// TIA Portal project "Phase 1" (V15.1)

(* hardware
DEVICE "S71500/ET200MP-Station_1"  S7-1500 station
   slot 0: "Profilschiene_0"  6ES7 590-1***0-0AA0
   slot 1: "PLC_1"  CPU 1511-1 PN  6ES7 511-1AK00-0AB0  V1.8
   slot 2: "AI 8xU/I/RTD/TC ST_1"  AI 8xU/I/RTD/TC ST  6ES7 531-7KF00-0AB0  V2.0
   slot 3: "AI 8xU/I/RTD/TC ST_2"  AI 8xU/I/RTD/TC ST  6ES7 531-7KF00-0AB0  V2.0
   slot 4: "AI 8xU/I/RTD/TC ST_3"  AI 8xU/I/RTD/TC ST  6ES7 531-7KF00-0AB0  V2.0
   slot 5: "AI 8xU/I/RTD/TC ST_4"  AI 8xU/I/RTD/TC ST  6ES7 531-7KF00-0AB0  V2.0
   slot 6: "DI 16x24VDC BA_1"  DI 16x24VDC BA  6ES7 521-1BH10-0AA0  V1.0
DEVICE "HMI_1"  KTP700 Basic PN
   slot 0: "HMI_1"  KTP700 Basic PN  6AV2 123-2GB03-0AX0  15.1.0.0
   slot 1: "HMI_RT_1"  KTP700 Basic PN  6AV2 123-2GB03-0AX0  15.1.0.0
   slot 5: "HMI_1.IE_CP_1"  PROFINET Interface  15.0.1.0
      slot 1: "PROFINET Interface_1"  PROFINET Interface
         slot 1: "Port_1"  Port
*)

// ===== PLC "PLC_1"  CPU 1511-1 PN =====

VAR_GLOBAL   // PLC tag table "Standard-Variablentabelle"
   "LevelMeter" AT %IW30 : Word;
   "FlowMeter" AT %IW32 : Word;
   "Set_point" AT %IW34 : Word;
   "Norm_SP" AT %MD74 : Real;
   "PID_Output" AT %MD104 : Real;
   "Start" AT %I10.0 : Bool;
   "Fill_Valve" AT %QW30 : Word;
   "Start_Light" AT %Q10.0 : Bool;
   "Reset" AT %I10.1 : Bool;
   "Reset_Light" AT %Q10.1 : Bool;
   "On" AT %M2.1 : Bool;
   "Stop" AT %I10.2 : Bool;
   "Stop_Light" AT %Q10.2 : Bool;
   "PV_display" AT %QW36 : Word;
   "Setpoint_display" AT %QW34 : Word;
   "Setpoint_value" AT %MD200 : Real;
   "Process_value" AT %MD204 : Real;
   "Norm_PID_Output" AT %MD208 : Real;
   "Start_from_HMI" AT %M4.0 : Bool;
   "Stop_from_HMI" AT %M4.1 : Bool;
   "Reset_from_HMI" AT %M4.2 : Bool;
   "Start_flag" AT %M5.0 : Bool;
   "Reset_flag" AT %M5.1 : Bool;
   "Stop_flag" AT %M5.2 : Bool;
   "Switch" AT %M5.3 : Bool;
   "Set_form_HMI" AT %MW216 : Word;
   "Norm_level" AT %MD212 : Real;
   "Level_error_margin" AT %MD218 : Real;
   "High_level_threshold" AT %MD220 : Real;
   "Low_level_threshold" AT %MD222 : Real;
   "Digital alarms" AT %MW6 : Word;
   "Discharge valve" AT %QW32 : Word;
END_VAR

// folder: System blocks/Program resources

DATA_BLOCK "IEC_Timer_0_DB"   // DB4
{ S7_Optimized_Access := 'TRUE' }
AUTHOR : Simatic
FAMILY : IEC
NAME : IEC_TMR
VERSION : 1.0
// stored: InstanceOfName IEC_TIMER
"IEC_TIMER"
BEGIN
END_DATA_BLOCK

// folder: (top level)

FUNCTION "MHJ-PLC-Lab-Function-S71500" : Void   // FC9000, SCL
{ S7_Optimized_Access := 'TRUE' }
VERSION : 0.1
   VAR_TEMP
      Value : Byte;
      ForCounter : Int;
   END_VAR
   VAR CONSTANT
      Value_01_DW : DWord := 16#1223_5486;
      Value_02_DW : DWord := 16#A6C9_D1F5;
   END_VAR
BEGIN

   #Value:=PEEK(area := 16#82,
        dbNumber := 0,
        byteOffset := 511);
   #Value := #Value + 1;

   POKE(area := 16#82,
        dbNumber := 0,
        byteOffset := 511,
        value := #Value);

   POKE(area := 16#82,
        dbNumber := 0,
        byteOffset := 1016,
        value := #Value_01_DW);
   POKE(area := 16#82,
        dbNumber := 0,
        byteOffset := 1020,
        value := #Value_02_DW);

   FOR #ForCounter := 0 TO 63 DO
       #Value:=PEEK(area := 16#1,
            dbNumber := 0,
            byteOffset := #ForCounter);
       POKE(area := 16#81,
            dbNumber := 0,
            byteOffset := #ForCounter,
            value := #Value);
   END_FOR;
   #Value := PEEK(area := 16#1,
                  dbNumber := 0,
                  byteOffset := 512);
   POKE(area := 16#82,
        dbNumber := 0,
        byteOffset := 512,
        value := #Value);
END_FUNCTION

ORGANIZATION_BLOCK "Main"   // OB1, FBD, ProgramCycle
TITLE = "Main Program Sweep (Cycle)"
{ S7_Optimized_Access := 'TRUE' }
VERSION : 0.1
   VAR_INPUT
      Initial_Call : Bool;   // Initial call of this OB
      Remanence : Bool;   // =True, if remanent data are available
   END_VAR
BEGIN

REGION Network 1
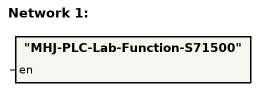
   "MHJ-PLC-Lab-Function-S71500"();
END_REGION
END_ORGANIZATION_BLOCK

ORGANIZATION_BLOCK "Cyclic interrupt"   // OB30, LAD, CyclicInterrupt
{ S7_Optimized_Access := 'TRUE' }
VERSION : 0.1
   VAR_INPUT
      Initial_Call : Bool;   // Initial call of this OB
      Event_Count : Int;   // Events discarded
   END_VAR
BEGIN

REGION Network 1
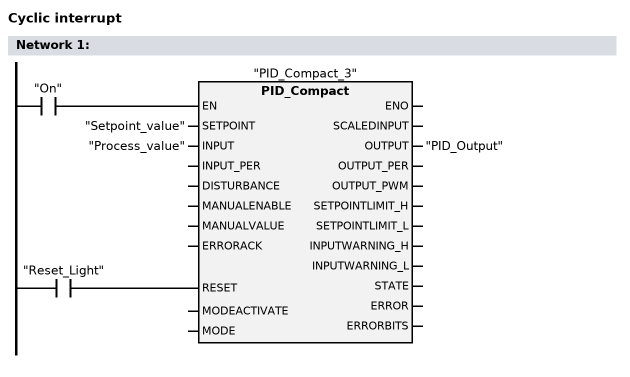
   IF "On" THEN
       "PID_Compact_3"(Setpoint := "Setpoint_value",   // PID_Compact
                       Input := "Process_value",
                       Reset := "Reset_Light",
                       Output => "PID_Output");
   END_IF;
END_REGION
END_ORGANIZATION_BLOCK

ORGANIZATION_BLOCK "Main_1"   // OB123, LAD, ProgramCycle
TITLE = "Main Program Sweep (Cycle)"
{ S7_Optimized_Access := 'TRUE' }
VERSION : 0.1
   VAR_INPUT
      Initial_Call : Bool;   // Initial call of this OB
      Remanence : Bool;   // =True, if remanent data are available
   END_VAR
BEGIN

REGION Network 1: Set point scale & display
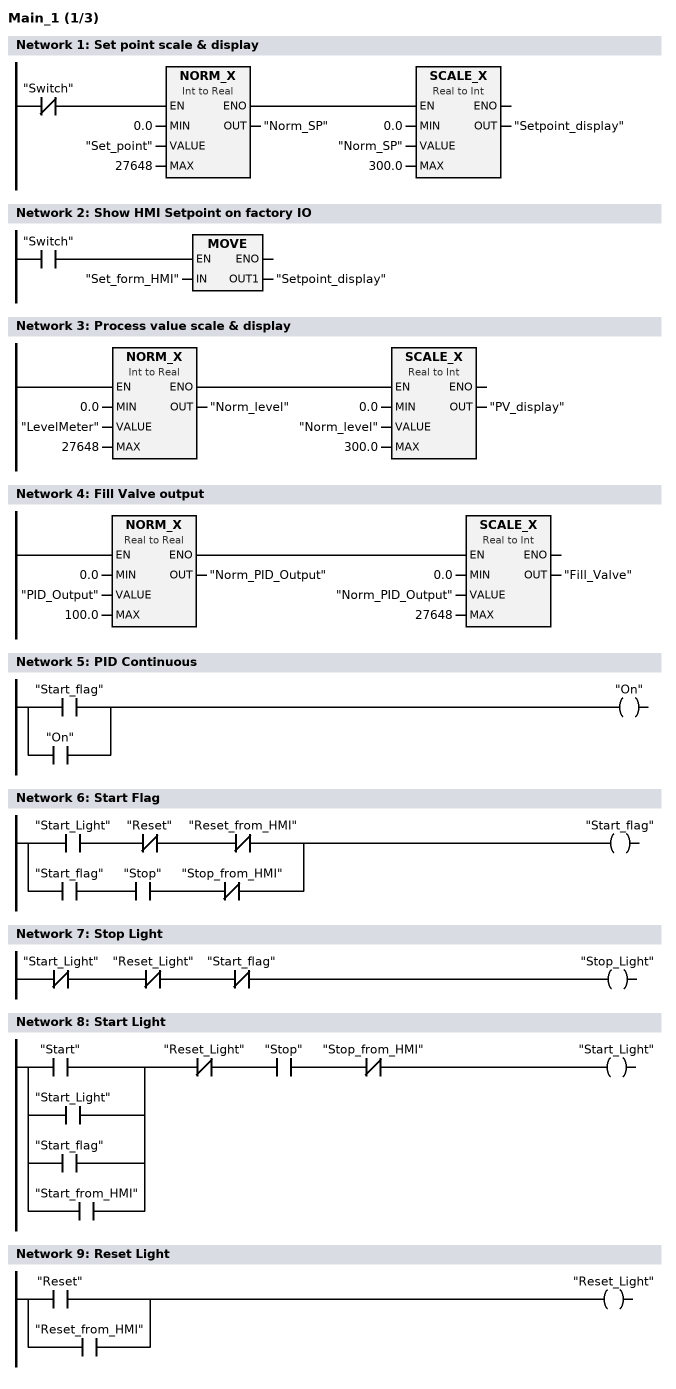
   RUNG wire#powerrail
      I_Contact( "Switch" )
      { S7_Templates := "[SrcType := Int, DestType := Real]" } Normalize(min := 0.0, value := "Set_point", max := 27648, out => "Norm_SP")
      { S7_Templates := "[SrcType := Real, DestType := Int]" } Scale(min := 0.0, value := "Norm_SP", max := 300.0, out => "Setpoint_display")
   END_RUNG
   // the same network as SCL:
   IF NOT "Switch" THEN
       "Norm_SP" := NORM_X(MIN := 0.0, VALUE := "Set_point", MAX := 27648);
       "Setpoint_display" := SCALE_X(MIN := 0.0, VALUE := "Norm_SP", MAX := 300.0);
   END_IF;
END_REGION

REGION Network 2: Show HMI Setpoint on factory IO
   RUNG wire#powerrail
      Contact( "Switch" )
      Move(in := "Set_form_HMI", out1 => "Setpoint_display")
   END_RUNG
   // the same network as SCL:
   IF "Switch" THEN "Setpoint_display" := "Set_form_HMI"; END_IF;
END_REGION

REGION Network 3: Process value scale & display
   RUNG wire#powerrail
      { S7_Templates := "[SrcType := Int, DestType := Real]" } Normalize(min := 0.0, value := "LevelMeter", max := 27648, out => "Norm_level")
      { S7_Templates := "[SrcType := Real, DestType := Int]" } Scale(min := 0.0, value := "Norm_level", max := 300.0, out => "PV_display")
   END_RUNG
   // the same network as SCL:
   "Norm_level" := NORM_X(MIN := 0.0, VALUE := "LevelMeter", MAX := 27648);
   "PV_display" := SCALE_X(MIN := 0.0, VALUE := "Norm_level", MAX := 300.0);
END_REGION

REGION Network 4: Fill Valve output
   RUNG wire#powerrail
      { S7_Templates := "[SrcType := Real, DestType := Real]" } Normalize(min := 0.0, value := "PID_Output", max := 100.0, out => "Norm_PID_Output")
      { S7_Templates := "[SrcType := Real, DestType := Int]" } Scale(min := 0.0, value := "Norm_PID_Output", max := 27648, out => "Fill_Valve")
   END_RUNG
   // the same network as SCL:
   "Norm_PID_Output" := NORM_X(MIN := 0.0, VALUE := "PID_Output", MAX := 100.0);
   "Fill_Valve" := SCALE_X(MIN := 0.0, VALUE := "Norm_PID_Output", MAX := 27648);
END_REGION

REGION Network 5: PID Continuous
   RUNG wire#powerrail
      Contact( "Start_flag" )
      wire#w1
      Coil( "On" )
   END_RUNG
   RUNG wire#powerrail
      Contact( "On" )
   END_RUNG wire#w1
   // the same network as SCL:
   "On" := "Start_flag" OR "On";
END_REGION

REGION Network 6: Start Flag
   RUNG wire#powerrail
      Contact( "Start_Light" )
      I_Contact( "Reset" )
      I_Contact( "Reset_from_HMI" )
      wire#w1
      Coil( "Start_flag" )
   END_RUNG
   RUNG wire#powerrail
      Contact( "Start_flag" )
      Contact( "Stop" )
      I_Contact( "Stop_from_HMI" )
   END_RUNG wire#w1
   // the same network as SCL:
   "Start_flag" := ("Start_Light" AND NOT "Reset" AND NOT "Reset_from_HMI") OR ("Start_flag" AND "Stop" AND NOT "Stop_from_HMI");
END_REGION

REGION Network 7: Stop Light
   RUNG wire#powerrail
      I_Contact( "Start_Light" )
      I_Contact( "Reset_Light" )
      I_Contact( "Start_flag" )
      Coil( "Stop_Light" )
   END_RUNG
   // the same network as SCL:
   "Stop_Light" := NOT "Start_Light" AND NOT "Reset_Light" AND NOT "Start_flag";
END_REGION

REGION Network 8: Start Light
   RUNG wire#powerrail
      Contact( "Start" )
      wire#w1
      I_Contact( "Reset_Light" )
      Contact( "Stop" )
      I_Contact( "Stop_from_HMI" )
      Coil( "Start_Light" )
   END_RUNG
   RUNG wire#powerrail
      Contact( "Start_Light" )
   END_RUNG wire#w1
   RUNG wire#powerrail
      Contact( "Start_flag" )
   END_RUNG wire#w1
   RUNG wire#powerrail
      Contact( "Start_from_HMI" )
   END_RUNG wire#w1
   // the same network as SCL:
   "Start_Light" := ("Start" OR "Start_Light" OR "Start_flag" OR "Start_from_HMI") AND NOT "Reset_Light" AND "Stop" AND NOT "Stop_from_HMI";
END_REGION

REGION Network 9: Reset Light
   RUNG wire#powerrail
      Contact( "Reset" )
      wire#w1
      Coil( "Reset_Light" )
   END_RUNG
   RUNG wire#powerrail
      Contact( "Reset_from_HMI" )
   END_RUNG wire#w1
   // the same network as SCL:
   "Reset_Light" := "Reset" OR "Reset_from_HMI";
END_REGION

REGION Network 10: Fill Valve Stop
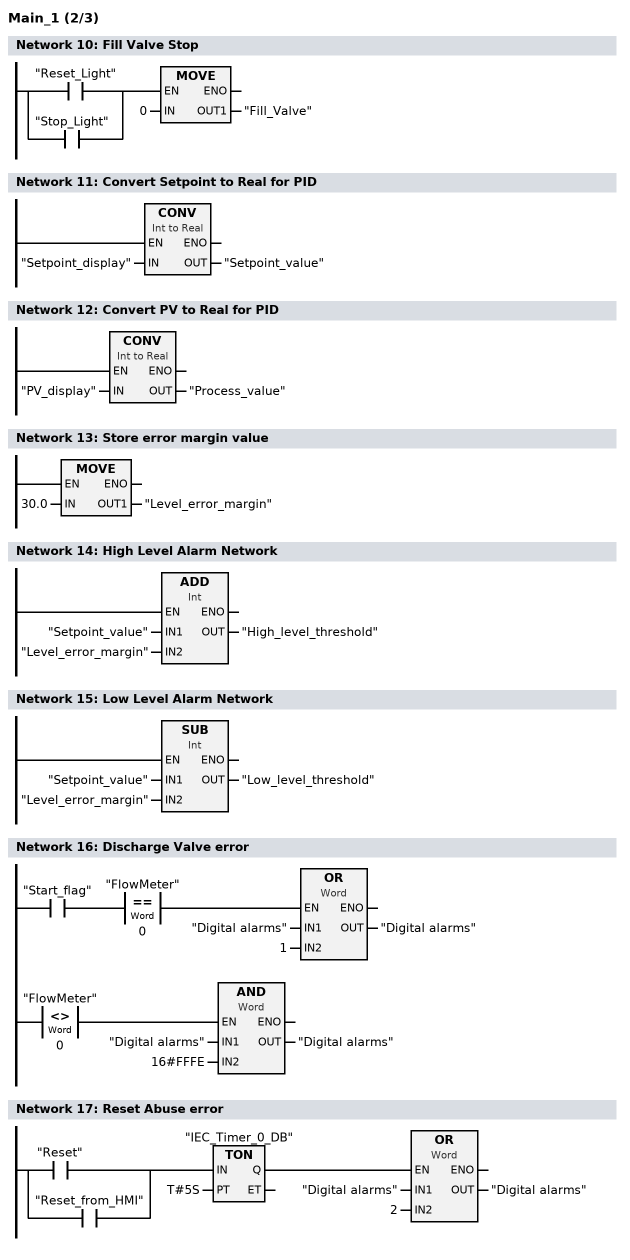
   RUNG wire#powerrail
      Contact( "Reset_Light" )
      wire#w1
      Move(in := 0, out1 => "Fill_Valve")
   END_RUNG
   RUNG wire#powerrail
      Contact( "Stop_Light" )
   END_RUNG wire#w1
   // the same network as SCL:
   IF "Reset_Light" OR "Stop_Light" THEN "Fill_Valve" := 0; END_IF;
END_REGION

REGION Network 11: Convert Setpoint to Real for PID
   RUNG wire#powerrail
      { S7_Templates := "[SrcType := Int, DestType := Real]" } Convert(in := "Setpoint_display", out => "Setpoint_value")
   END_RUNG
   // the same network as SCL:
   "Setpoint_value" := INT_TO_REAL("Setpoint_display");
END_REGION

REGION Network 12: Convert PV to Real for PID
   RUNG wire#powerrail
      { S7_Templates := "[SrcType := Int, DestType := Real]" } Convert(in := "PV_display", out => "Process_value")
   END_RUNG
   // the same network as SCL:
   "Process_value" := INT_TO_REAL("PV_display");
END_REGION

REGION Network 13: Store error margin value
   RUNG wire#powerrail
      Move(in := 30.0, out1 => "Level_error_margin")
   END_RUNG
   // the same network as SCL:
   "Level_error_margin" := 30.0;
END_REGION

REGION Network 14: High Level Alarm Network
   RUNG wire#powerrail
      { S7_Templates := "SrcType := Int" } Add(in1 := "Setpoint_value", in2 := "Level_error_margin", out => "High_level_threshold")
   END_RUNG
   // the same network as SCL:
   "High_level_threshold" := "Setpoint_value" + "Level_error_margin";
END_REGION

REGION Network 15: Low Level Alarm Network
   RUNG wire#powerrail
      { S7_Templates := "SrcType := Int" } Sub(in1 := "Setpoint_value", in2 := "Level_error_margin", out => "Low_level_threshold")
   END_RUNG
   // the same network as SCL:
   "Low_level_threshold" := "Setpoint_value" - "Level_error_margin";
END_REGION

REGION Network 16: Discharge Valve error
   IF "Start_flag" AND ("FlowMeter" = 0) THEN "Digital alarms" := "Digital alarms" OR 1; END_IF;
   IF "FlowMeter" <> 0 THEN "Digital alarms" := "Digital alarms" AND 16#FFFE; END_IF;
END_REGION

REGION Network 17: Reset Abuse error
   "IEC_Timer_0_DB".TON(IN := "Reset" OR "Reset_from_HMI", PT := T#5S);
   IF "IEC_Timer_0_DB".Q THEN "Digital alarms" := "Digital alarms" OR 2; END_IF;
END_REGION

REGION Network 18: Reset Abuse error reset
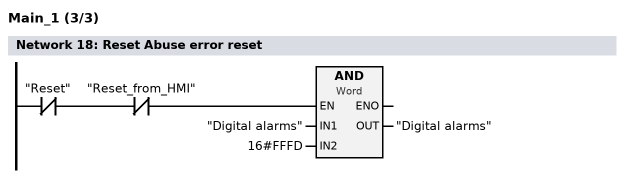
   RUNG wire#powerrail
      I_Contact( "Reset" )
      I_Contact( "Reset_from_HMI" )
      { S7_Templates := "SrcType := Word" } And(in1 := "Digital alarms", in2 := 16#FFFD, out => "Digital alarms")
   END_RUNG
   // the same network as SCL:
   IF NOT "Reset" AND NOT "Reset_from_HMI" THEN "Digital alarms" := "Digital alarms" AND 16#FFFD; END_IF;
END_REGION
END_ORGANIZATION_BLOCK

(* ===== HMI "HMI_RT_1" =====
system functions are stored by id; their names below are inferred from use
connection "HMI_Connection_1": ETHERNET, SMART_S7_1500_OMS

HMI tags "Default tag table"
   "Tag_ScreenNumber" : UInt, internal
   "Start_from_HMI" : Bool = PLC Start_from_HMI AT %M4.0, 1 s
   "Stop_from_HMI" : Bool = PLC Stop_from_HMI AT %M4.1, 1 s
   "Reset_from_HMI" : Bool = PLC Reset_from_HMI AT %M4.2, 1 s
   "Start_Light" : Bool = PLC Start_Light AT %Q10.0, 1 s
   "Stop_Light" : Bool = PLC Stop_Light AT %Q10.2, 1 s
   "Reset_Light" : Bool = PLC Reset_Light AT %Q10.1, 1 s
   "PV_display" : Word = PLC PV_display AT %QW36, 1 s
   "Setpoint_display" : Word = PLC Setpoint_display AT %QW34, 1 s
   "Set_point" : Word = PLC Set_point AT %IW34, 1 s
   "Switch" : Bool = PLC Switch AT %M5.3, 1 s
   "Set_form_HMI" : Word = PLC Set_form_HMI AT %MW216, 1 s
   "Process_value" : Real = PLC Process_value AT %MD204, 1 s
   "Setpoint_value" : Real = PLC Setpoint_value AT %MD200, 1 s
   "High_level_threshold" : Real = PLC High_level_threshold AT %MD220, 1 s
   "Low_level_threshold" : Real = PLC Low_level_threshold AT %MD222, 1 s
   "Level_error_margin" : Real = PLC Level_error_margin AT %MD218, 1 s
   "Digital alarms" : Word = PLC "Digital alarms" AT %MW6, 1 s

discrete alarms
   1004: 'Discharge valve is either clogged , or not operating as required , please check!', class Warnings, trigger "Digital alarms" bit 0
   1005: 'Reset Button is pressed for a long time , please check.', class Warnings, trigger "Digital alarms" bit 1

analog alarms
   1000: 'Liquid level reached critical high level!', class Errors, trigger "PV_display"
   1001: 'Liquid level reached critical low level level!', class Errors, trigger "PV_display"
   1002: 'Liquid level is higher than setpoint , if warning didnt disappear , check flow rate or sensor readings.', class Warnings, trigger "PV_display"
   1003: 'Liquid Level is lower than setpoint , if warning didnt disappear , check flow rate or sensor readings.', class Warnings, trigger "PV_display"

Template "Template_1" 800x480
   Button "Exit" at 714,429 size 71x50; TextOff 'Exit'; PictureOff "ExitRuntime_KTP700_Basic_PN_TR"; PictureOn "ExitRuntime_KTP700_Basic_PN_TR"
      on Release: StopRuntime(0)
   Button "Template_Button" at 614,429 size 71x50; TextOff 'Text'
   Button "Template_Button_1" at 514,429 size 71x50; TextOff 'Text'
   Button "Template_Button_2" at 414,429 size 71x50; TextOff 'Text'
   Button "Template_Button_3" at 314,429 size 71x50; TextOff 'Text'
   Button "Template_Button_4" at 214,429 size 71x50; TextOff 'Text'
   Button "Alarms" at 114,429 size 71x50; TextOff 'Alarms'; PictureOff "AlarmDisplay_KTP700_Basic_PN_TR"; PictureOn "AlarmDisplay_KTP700_Basic_PN_TR"
      on Release: function_ef3f5d25("Alarm window_Unacknowledged", -1)
   Button "Start screen" at 14,429 size 71x50; TextOff 'Start screen'; PictureOff "NavigateHome_KTP700_Basic_PN_TR"; PictureOn "NavigateHome_KTP700_Basic_PN_TR"
      on Release: ActivateScreen("Root screen", 0)
   SymbolicIOField "Symbolic_IO_Field_Screen" at 93,9 size 600x33; TextOff '0'; TextOn '1'; TextList "TextList_ScreenNames"
      ProcessValue <- "Tag_ScreenNumber"
      on Change: ActivateScreenByNumber("Tag_ScreenNumber", 0)
   DateTimeField "HmiScreenItemData" at 695,25 size 105x25
   DateTimeField "HmiScreenItemData_1" at 695,0 size 105x25
   GraphicView "Logo" at 0,0 size 91x51; Picture "Logo of HMI_1"

screen "Root screen" 800x480, template "Template_1"
   on GenerateScreen: SetTag("Tag_ScreenNumber", 1)
   GraphicView "Graphic view_1" at 0,50 size 800x430; Picture "robot-machine-engineering-factory-wallpaper-preview"
   TextField "HmiScreenItemData_1" at 297,57 size 196x30; Text 'Welcome to phase one'
   Button "Button_1" at 87,432 size 96x32; TextOff 'Start'
      on Press: function_b14e0dd5("Start_from_HMI", 0)
   Button "Button_2" at 349,432 size 96x32; TextOff 'Stop'
      on Press: function_b14e0dd5("Stop_from_HMI", 0)
   Button "Button_3" at 623,432 size 96x32; TextOff 'Reset'
      on Press: function_b14e0dd5("Reset_from_HMI", 0)
   Circle "Circle_1" at 112,376 size 48x48
      Appearance <- "Start_Light"
   Circle "Circle_2" at 371,376 size 48x48
      Appearance <- "Stop_Light"
   Circle "Circle_3" at 645,376 size 48x48
      Appearance <- "Reset_Light"
   AlarmView "Alarm view_1" at 17,92 size 426x279
   IOField "I/O field_2" at 634,74 size 96x32; FormatPattern 999
      ProcessValue <- "Process_value"
   IOField "I/O field_1" at 491,106 size 96x32; FormatPattern 999
      ProcessValue <- "Set_form_HMI"
   TextField "Text field_3" at 498,147 size 80x23; Text 'Set Point'
   Switch "Switch_1" at 507,251 size 64x32; CaptionText 'Switch'; TextOff 'OFF'; TextOn 'ON'
      ProcessValue <- "Switch"
   TextField "Text field_2" at 483,289 size 111x23; Text 'Take Control'
   TextField "Text field_1" at 636,338 size 94x23; Text 'Tank Level'
   Bar "Bar_1" at 643,113 size 79x215; MinimumValue 0; MaximumValue 300
      ProcessValue <- "PV_display"

screen "PID trend" 800x480, template "Template_1"
   on GenerateScreen: SetTag("Tag_ScreenNumber", 2)
   TextField "HmiScreenItemData" at 80,225 size 640x25; Text 'PID trend'
   TrendView "Trend view_1" at 0,49 size 800x431
*)